PROGRAM S3_01_Motion_2
VAR
	HMI_Motion: FB_HMI_Control;
	Motion: FB_Motion2way;

	tMessageOffset: UINT;
	tNumMessagesPerRow: UINT;
	
	
	MyAdvanceInterlock: BOOL;
	MyReturnInterlock: BOOL;
	
	MyAutoAdvanceCondition: BOOL;
	MyAutoReturnCondition: BOOL;
	testword: WORD;
	myAdvancePrompt: BOOL;
	myReturnPrompt: BOOL;
	advancedSensor: BOOL;
	returnedSensor: BOOL;
	AdvanceCoil: BOOL;
	ReturnCoil: BOOL;
	tWaitMsgXICAdv: BOOL;
	tWaitMsgXICRet: BOOL;
END_VAR

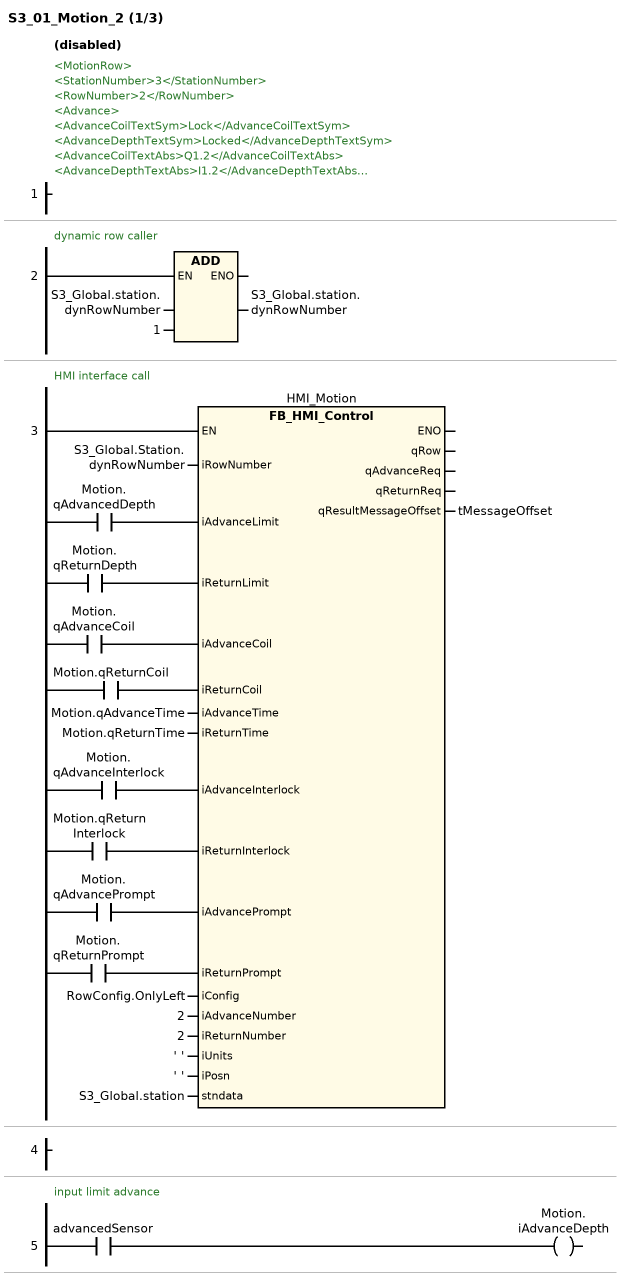
// NETWORK 1 (disabled)
// <MotionRow>
// <StationNumber>3</StationNumber>
// <RowNumber>2</RowNumber>
//   <Advance>
//     <AdvanceCoilTextSym>Lock</AdvanceCoilTextSym>
//     <AdvanceDepthTextSym>Locked</AdvanceDepthTextSym>
//     <AdvanceCoilTextAbs>Q1.2</AdvanceCoilTextAbs>
//     <AdvanceDepthTextAbs>I1.2</AdvanceDepthTextAbs>
//     <ManSeq>3</ManSeq>
//   </Advance>
//   <Return>
//     <ReturnCoilTextSym>Unlock</ReturnCoilTextSym>
//     <ReturnDepthTextSym>Unlocked</ReturnDepthTextSym>
//     <ReturnCoilTextAbs>Q1.3</ReturnCoilTextAbs>
//     <ReturnDepthTextAbs>I1.3</ReturnDepthTextAbs>
//    <ManSeq>4</ManSeq>
//   </Return>
//   <Motion>
//     <NameSym>Lock Cylinder</NameSym>
//     <NameAbs>A2</NameAbs>
//   </Motion>
// </MotionRow>

// NETWORK 2
// dynamic row caller
S3_Global.station.dynRowNumber := S3_Global.station.dynRowNumber + 1;

// NETWORK 3
// HMI interface call
HMI_Motion(
    iRowNumber := S3_Global.Station.dynRowNumber,
    iAdvanceLimit := Motion.qAdvancedDepth,
    iReturnLimit := Motion.qReturnDepth,
    iAdvanceCoil := Motion.qAdvanceCoil,
    iReturnCoil := Motion.qReturnCoil,
    iAdvanceTime := Motion.qAdvanceTime,
    iReturnTime := Motion.qReturnTime,
    iAdvanceInterlock := Motion.qAdvanceInterlock,
    iReturnInterlock := Motion.qReturnInterlock,
    iAdvancePrompt := Motion.qAdvancePrompt,
    iReturnPrompt := Motion.qReturnPrompt,
    iConfig := RowConfig.OnlyLeft,
    iAdvanceNumber := 2,
    iReturnNumber := 2,
    iUnits := ' ',
    iPosn := ' ',
    stndata := S3_Global.station,
    qResultMessageOffset => tMessageOffset); // FB_HMI_Control

// NETWORK 4

// NETWORK 5
// input limit advance
Motion.iAdvanceDepth := advancedSensor;

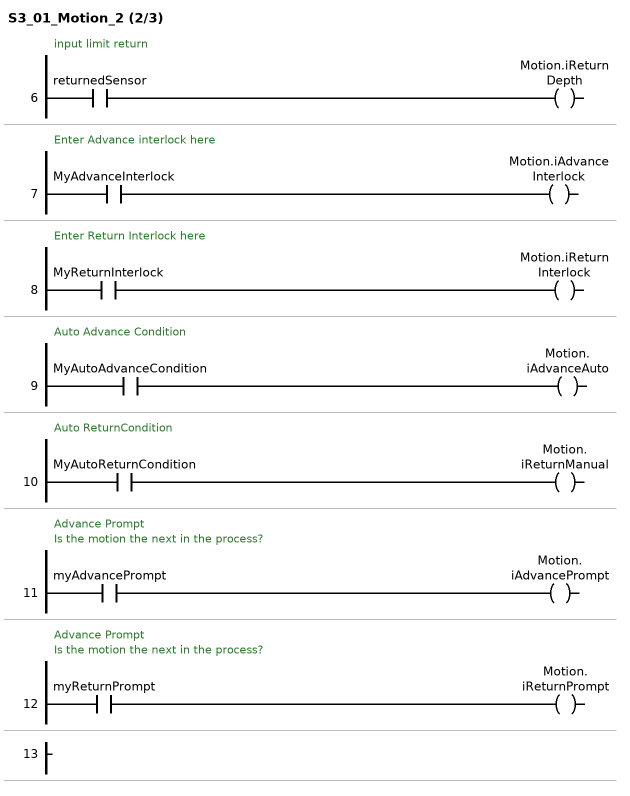
// NETWORK 6
// input limit return
Motion.iReturnDepth := returnedSensor;

// NETWORK 7
// Enter Advance interlock here
Motion.iAdvanceInterlock := MyAdvanceInterlock;

// NETWORK 8
// Enter Return Interlock here
Motion.iReturnInterlock := MyReturnInterlock;

// NETWORK 9
// Auto Advance Condition
Motion.iAdvanceAuto := MyAutoAdvanceCondition;

// NETWORK 10
// Auto ReturnCondition
Motion.iReturnManual := MyAutoReturnCondition;

// NETWORK 11
// Advance Prompt
// Is the motion the next in the process?
Motion.iAdvancePrompt := myAdvancePrompt;

// NETWORK 12
// Advance Prompt
// Is the motion the next in the process?
Motion.iReturnPrompt := myReturnPrompt;

// NETWORK 13

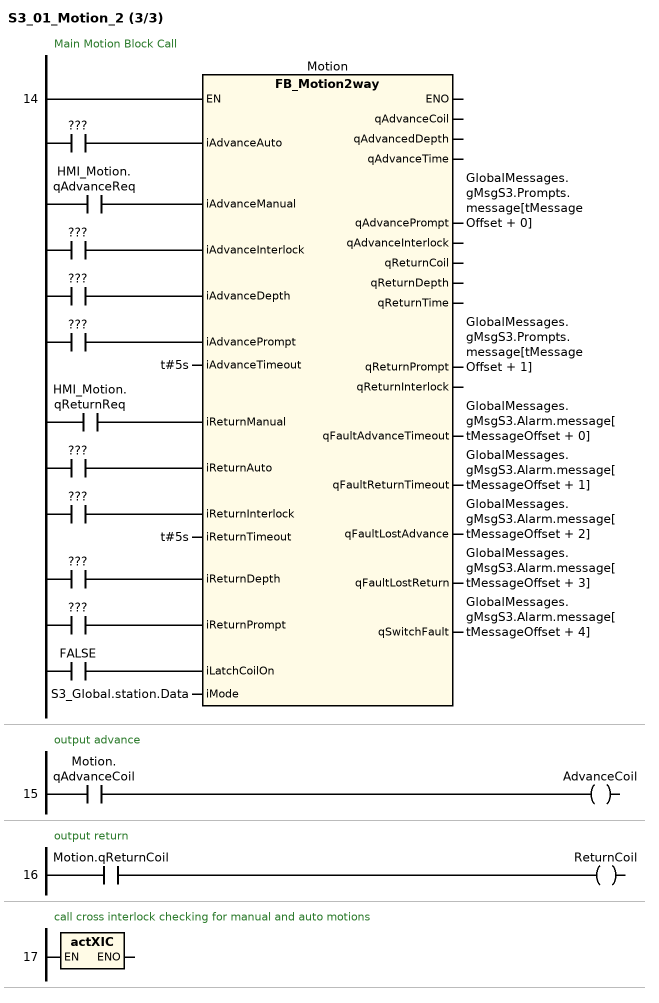
// NETWORK 14
// Main Motion Block Call
Motion(
    iAdvanceManual := HMI_Motion.qAdvanceReq,
    iAdvanceTimeout := t#5s,
    iReturnManual := HMI_Motion.qReturnReq,
    iReturnTimeout := t#5s,
    iLatchCoilOn := FALSE,
    iMode := S3_Global.station.Data,
    qAdvancePrompt => GlobalMessages.gMsgS3.Prompts.message[tMessageOffset + 0],
    qReturnPrompt => GlobalMessages.gMsgS3.Prompts.message[tMessageOffset + 1],
    qFaultAdvanceTimeout => GlobalMessages.gMsgS3.Alarm.message[tMessageOffset + 0],
    qFaultReturnTimeout => GlobalMessages.gMsgS3.Alarm.message[tMessageOffset + 1],
    qFaultLostAdvance => GlobalMessages.gMsgS3.Alarm.message[tMessageOffset + 2],
    qFaultLostReturn => GlobalMessages.gMsgS3.Alarm.message[tMessageOffset + 3],
    qSwitchFault => GlobalMessages.gMsgS3.Alarm.message[tMessageOffset + 4]); // FB_Motion2way

// NETWORK 15
// output advance
AdvanceCoil := Motion.qAdvanceCoil;

// NETWORK 16
// output return
ReturnCoil := Motion.qReturnCoil;

// NETWORK 17
// call cross interlock checking for manual and auto motions
actXIC();

ACTION actXIC:
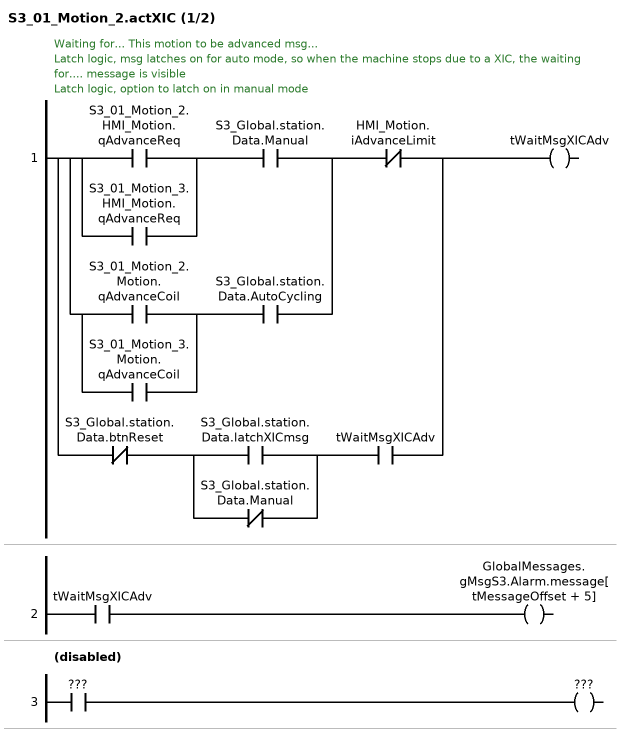
// NETWORK 1
// Waiting for... This motion to be advanced msg...
// Latch logic, msg latches on for auto mode, so when the machine stops due to a XIC, the waiting for.... message is visible
// Latch logic, option to latch on in manual mode
tWaitMsgXICAdv := ((S3_01_Motion_2.HMI_Motion.qAdvanceReq OR S3_01_Motion_3.HMI_Motion.qAdvanceReq) AND S3_Global.station.Data.Manual OR (S3_01_Motion_2.Motion.qAdvanceCoil OR S3_01_Motion_3.Motion.qAdvanceCoil) AND S3_Global.station.Data.AutoCycling) AND NOT HMI_Motion.iAdvanceLimit OR NOT S3_Global.station.Data.btnReset AND (S3_Global.station.Data.latchXICmsg OR NOT S3_Global.station.Data.Manual) AND tWaitMsgXICAdv;

// NETWORK 2
GlobalMessages.gMsgS3.Alarm.message[tMessageOffset + 5] := tWaitMsgXICAdv;

// NETWORK 3 (disabled)
// ??? := ???;

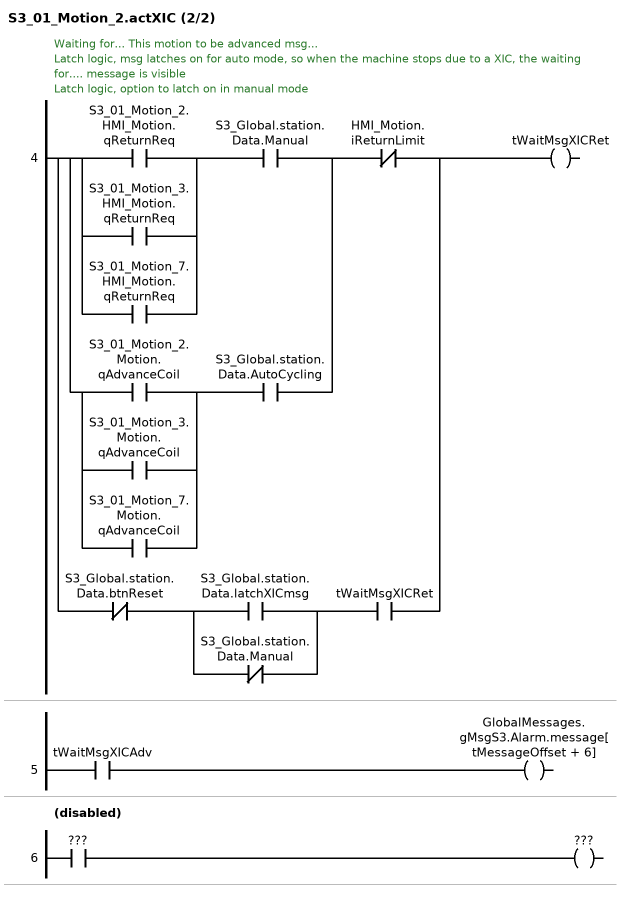
// NETWORK 4
// Waiting for... This motion to be advanced msg...
// Latch logic, msg latches on for auto mode, so when the machine stops due to a XIC, the waiting for.... message is visible
// Latch logic, option to latch on in manual mode
tWaitMsgXICRet := ((S3_01_Motion_2.HMI_Motion.qReturnReq OR S3_01_Motion_3.HMI_Motion.qReturnReq OR S3_01_Motion_7.HMI_Motion.qReturnReq) AND S3_Global.station.Data.Manual OR (S3_01_Motion_2.Motion.qAdvanceCoil OR S3_01_Motion_3.Motion.qAdvanceCoil OR S3_01_Motion_7.Motion.qAdvanceCoil) AND S3_Global.station.Data.AutoCycling) AND NOT HMI_Motion.iReturnLimit OR NOT S3_Global.station.Data.btnReset AND (S3_Global.station.Data.latchXICmsg OR NOT S3_Global.station.Data.Manual) AND tWaitMsgXICRet;

// NETWORK 5
GlobalMessages.gMsgS3.Alarm.message[tMessageOffset + 6] := tWaitMsgXICAdv;

// NETWORK 6 (disabled)
// ??? := ???;
END_ACTION

END_PROGRAM

(* stored: Version 1.1.0.1, ProductVersion 3.1.4024.11
   POU S3_01_Motion_2: Id {593529f4-7264-054e-12f5-af644d8b02c6}, SpecialFunc None
   Action actXIC: Id {d97381cd-0bf8-05a5-397b-1abaa59a781c} *)
